TYPE "PLCtoMES_AlarmMassage_ext"
VERSION : 0.1
   STRUCT
      "MES.ErrorCode" : Int;
      "MES.ErrorMsg" : String[60];
   END_STRUCT;

END_TYPE

